// TIA Portal V20 export
TYPE "typeCmControlNodeCommand"
// stored: Namespace Unit1.Em3
   STRUCT
      topTapeAxisX : "LER_typeAxisCommand";
      topTapeAxisY : "LER_typeAxisCommand";
      topTapeLoading { S7_SetPoint := 'True'} : "LER_typeTwoWayActCommand";
      topTapeLoadingClamp { S7_SetPoint := 'True'} : "LER_typeTwoWayActCommand";
      topTapeCutter { S7_SetPoint := 'True'} : "LER_typeTwoWayActCommand";
      topTapeCutterClamp { S7_SetPoint := 'True'} : "LER_typeTwoWayActCommand";
      topTapeTension { S7_SetPoint := 'True'} : "LER_typeTwoWayActCommand";
      topTapeAttachment { S7_SetPoint := 'True'} : "LER_typeTwoWayActCommand";
      topTapeClampTopLeft { S7_SetPoint := 'True'} : "LER_typeTwoWayActCommand";
      topTapeClampTopCenter { S7_SetPoint := 'True'} : "LER_typeTwoWayActCommand";
      topTapeClampTopRight { S7_SetPoint := 'True'} : "LER_typeTwoWayActCommand";
      topTapeClampBtm { S7_SetPoint := 'True'} : "LER_typeTwoWayActCommand";
      topTapeClampAll { S7_SetPoint := 'True'} : "LER_typeTwoWayActCommand";
      topTapeAttachmentVaccum { S7_SetPoint := 'True'} : "LER_typeTwoWayActCommand";
   END_STRUCT;
END_TYPE
